FUNCTION_BLOCK RASPBERRY_PI_CONTROL_ROBOT
  {SET_ATTRIBUTE(OpcUa, DEVICE.SENSOR)}
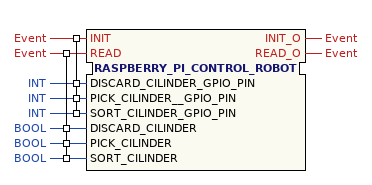
  EVENT_INPUT
    INIT WITH DISCARD_CILINDER_GPIO_PIN, PICK_CILINDER__GPIO_PIN, SORT_CILINDER_GPIO_PIN;
    READ WITH DISCARD_CILINDER, PICK_CILINDER, SORT_CILINDER;
  END_EVENT
  EVENT_OUTPUT
    INIT_O;
    READ_O;
  END_EVENT
  VAR_INPUT
    DISCARD_CILINDER_GPIO_PIN : INT; {SET_ATTRIBUTE(OpcUa, Constant.RUN)}
    PICK_CILINDER__GPIO_PIN : INT; {SET_ATTRIBUTE(OpcUa, Constant.RUN)}
    SORT_CILINDER_GPIO_PIN : INT; {SET_ATTRIBUTE(OpcUa, Constant.RUN)}
    DISCARD_CILINDER : BOOL; {SET_ATTRIBUTE(OpcUa, Variable.RUN)}
    PICK_CILINDER : BOOL; {SET_ATTRIBUTE(OpcUa, Variable.RUN)}
    SORT_CILINDER : BOOL; {SET_ATTRIBUTE(OpcUa, Variable.RUN)}
  END_VAR
END_FUNCTION_BLOCK
